// TIA Portal project "DistributionMPS" (V16)

(* hardware
DEVICE "S7-1200 station_1"  S7-1200 Station
   slot 0: "Rack_0"  S7-1200 Rack  Rack  V1.0
   slot 1: "PLC_1"  CPU 1214C AC/DC/Rly  6ES7 214-1BG31-0XB0  V3.0
DEVICE "HMI_1"  KTP600 Basic color PN
   slot 0: "HMI_1"  KTP600 Basic color PN  6AV6 647-0AD11-3AX0  12.0.0.0
   slot 1: "HMI_RT_1"  KTP600 Basic color PN  6AV6 647-0AD11-3AX0  12.0.0.0
   slot 5: "HMI_1.IE_CP_1"  PROFINET Interface  12.0.0.0
      slot 1: "Interfaz PROFINET_1"  PROFINET Interface
         slot 1: "Port_1"  Port
*)

// ===== PLC "PLC_1"  CPU 1214C AC/DC/Rly =====

VAR_GLOBAL   // PLC tag table "Tabla de variables estándar"
   "Conveyor_Forward" AT %Q0.0 : Bool;
   "Conveyor_Reverse" AT %Q0.1 : Bool;
   "Splitter" AT %Q0.2 : Bool;
   "Slider" AT %Q0.4 : Bool;
   "WP_Beg" AT %I0.0 : Bool;
   "WP_Mid" AT %I0.1 : Bool;
   "No_WP_End" AT %I0.2 : Bool;
   "Slider_Init" AT %I0.4 : Bool;
   "Slider_End" AT %I0.5 : Bool;
   "Mag_Empty" AT %I0.6 : Bool;
   "System_Ready" AT %M0.0 : Bool;
   "WP_In" AT %M0.1 : Bool;
   "WP_Eject" AT %M0.2 : Bool;
   "WP_In_Conveyor" AT %M0.3 : Bool;
   "No_WP_In_Mag" AT %M0.4 : Bool;
   "WP_Ej_Conveyor" AT %M0.5 : Bool;
END_VAR

// folder: System blocks/Program resources

DATA_BLOCK "IEC_Timer_0_DB"   // DB1
{ S7_Optimized_Access := 'TRUE' }
AUTHOR : Simatic
FAMILY : IEC
NAME : IEC_TMR
VERSION : 1.0
// stored: InstanceOfName IEC_TIMER
"IEC_TIMER"
BEGIN
END_DATA_BLOCK

DATA_BLOCK "IEC_Timer_0_DB_1"   // DB2
{ S7_Optimized_Access := 'TRUE' }
AUTHOR : Simatic
FAMILY : IEC
NAME : IEC_TMR
VERSION : 1.0
// stored: InstanceOfName IEC_TIMER
"IEC_TIMER"
BEGIN
END_DATA_BLOCK

// folder: (top level)

ORGANIZATION_BLOCK "Main"   // OB1, LAD, ProgramCycle
TITLE = "Main Program Sweep (Cycle)"
{ S7_Optimized_Access := 'TRUE' }
VERSION : 0.1
   VAR_TEMP   // added for the SCL form of the ladder/FBD networks
      _w1 : Bool;
   END_VAR
BEGIN

REGION Network 1: Identificar Pieza
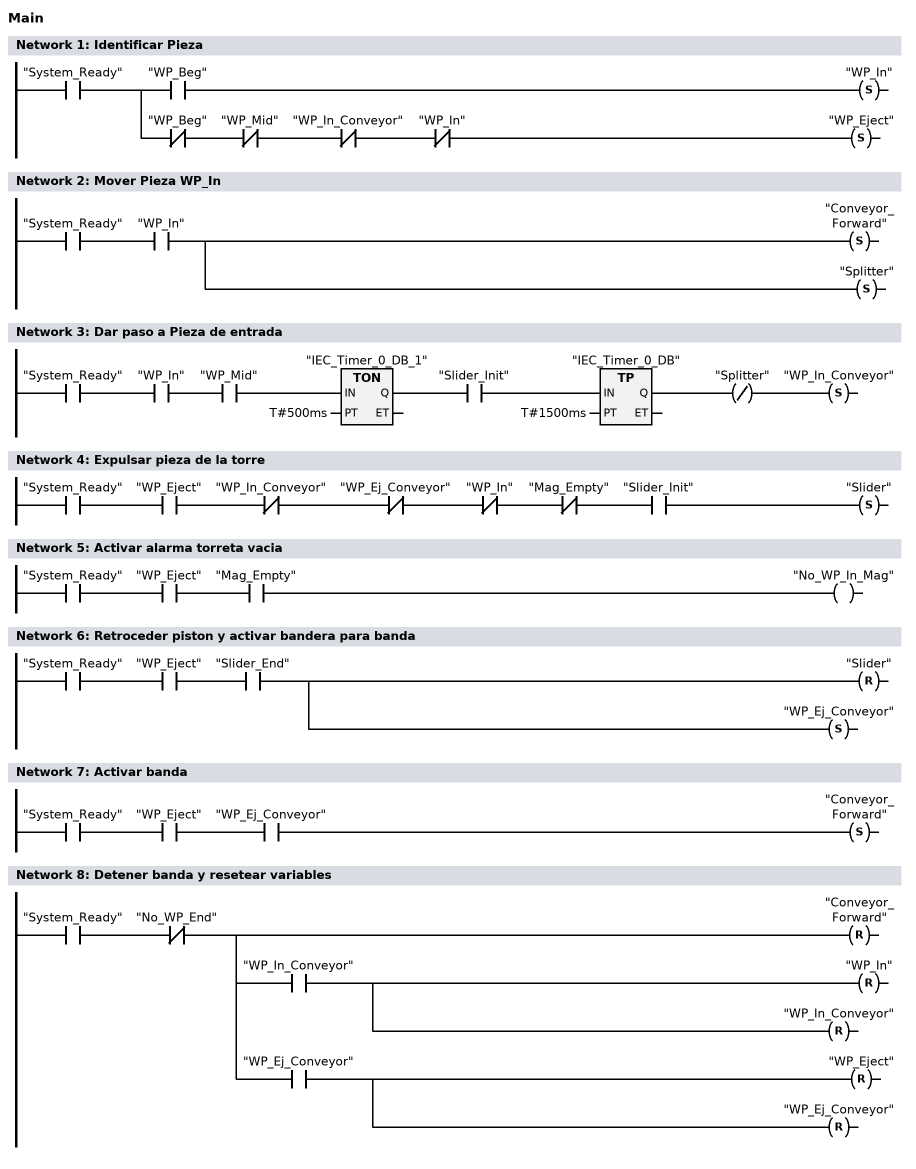
   RUNG wire#powerrail
      Contact( "System_Ready" )
      wire#w1
      Contact( "WP_Beg" )
      S_Coil( "WP_In" )
   END_RUNG
   RUNG wire#w1
      I_Contact( "WP_Beg" )
      I_Contact( "WP_Mid" )
      I_Contact( "WP_In_Conveyor" )
      I_Contact( "WP_In" )
      S_Coil( "WP_Eject" )
   END_RUNG
   // the same network as SCL:
   IF "System_Ready" AND "WP_Beg" THEN "WP_In" := TRUE; END_IF;
   IF "System_Ready" AND NOT "WP_Beg" AND NOT "WP_Mid" AND NOT "WP_In_Conveyor" AND NOT "WP_In" THEN
       "WP_Eject" := TRUE;
   END_IF;
END_REGION

REGION Network 2: Mover Pieza WP_In
   RUNG wire#powerrail
      Contact( "System_Ready" )
      Contact( "WP_In" )
      wire#w1
      S_Coil( "Conveyor_Forward" )
   END_RUNG
   RUNG wire#w1
      S_Coil( "Splitter" )
   END_RUNG
   // the same network as SCL:
   IF "System_Ready" AND "WP_In" THEN
       "Conveyor_Forward" := TRUE;
       "Splitter" := TRUE;
   END_IF;
END_REGION

REGION Network 3: Dar paso a Pieza de entrada
   "IEC_Timer_0_DB_1".TON(IN := "System_Ready" AND "WP_In" AND "WP_Mid", PT := T#500ms);
   "IEC_Timer_0_DB".TP(IN := "IEC_Timer_0_DB_1".Q AND "Slider_Init", PT := T#1500ms);
   "Splitter" := NOT "IEC_Timer_0_DB".Q;
   IF "IEC_Timer_0_DB".Q THEN "WP_In_Conveyor" := TRUE; END_IF;
END_REGION

REGION Network 4: Expulsar pieza de la torre
   RUNG wire#powerrail
      Contact( "System_Ready" )
      Contact( "WP_Eject" )
      I_Contact( "WP_In_Conveyor" )
      I_Contact( "WP_Ej_Conveyor" )
      I_Contact( "WP_In" )
      I_Contact( "Mag_Empty" )
      Contact( "Slider_Init" )
      S_Coil( "Slider" )
   END_RUNG
   // the same network as SCL:
   IF "System_Ready" AND "WP_Eject" AND NOT "WP_In_Conveyor" AND NOT "WP_Ej_Conveyor" AND NOT "WP_In" AND NOT "Mag_Empty" AND "Slider_Init" THEN
       "Slider" := TRUE;
   END_IF;
END_REGION

REGION Network 5: Activar alarma torreta vacia
   RUNG wire#powerrail
      Contact( "System_Ready" )
      Contact( "WP_Eject" )
      Contact( "Mag_Empty" )
      Coil( "No_WP_In_Mag" )
   END_RUNG
   // the same network as SCL:
   "No_WP_In_Mag" := "System_Ready" AND "WP_Eject" AND "Mag_Empty";
END_REGION

REGION Network 6: Retroceder piston y activar bandera para banda
   RUNG wire#powerrail
      Contact( "System_Ready" )
      Contact( "WP_Eject" )
      Contact( "Slider_End" )
      wire#w1
      R_Coil( "Slider" )
   END_RUNG
   RUNG wire#w1
      S_Coil( "WP_Ej_Conveyor" )
   END_RUNG
   // the same network as SCL:
   IF "System_Ready" AND "WP_Eject" AND "Slider_End" THEN
       "Slider" := FALSE;
       "WP_Ej_Conveyor" := TRUE;
   END_IF;
END_REGION

REGION Network 7: Activar banda
   RUNG wire#powerrail
      Contact( "System_Ready" )
      Contact( "WP_Eject" )
      Contact( "WP_Ej_Conveyor" )
      S_Coil( "Conveyor_Forward" )
   END_RUNG
   // the same network as SCL:
   IF "System_Ready" AND "WP_Eject" AND "WP_Ej_Conveyor" THEN "Conveyor_Forward" := TRUE; END_IF;
END_REGION

REGION Network 8: Detener banda y resetear variables
   RUNG wire#powerrail
      Contact( "System_Ready" )
      I_Contact( "No_WP_End" )
      wire#w1
      R_Coil( "Conveyor_Forward" )
   END_RUNG
   RUNG wire#w1
      Contact( "WP_In_Conveyor" )
      wire#w2
      R_Coil( "WP_In" )
   END_RUNG
   RUNG wire#w2
      R_Coil( "WP_In_Conveyor" )
   END_RUNG
   RUNG wire#w1
      Contact( "WP_Ej_Conveyor" )
      wire#w3
      R_Coil( "WP_Eject" )
   END_RUNG
   RUNG wire#w3
      R_Coil( "WP_Ej_Conveyor" )
   END_RUNG
   // the same network as SCL:
   #_w1 := "System_Ready" AND NOT "No_WP_End";
   IF #_w1 THEN "Conveyor_Forward" := FALSE; END_IF;
   IF #_w1 AND "WP_In_Conveyor" THEN
       "WP_In" := FALSE;
       "WP_In_Conveyor" := FALSE;
   END_IF;
   IF #_w1 AND "WP_Ej_Conveyor" THEN
       "WP_Eject" := FALSE;
       "WP_Ej_Conveyor" := FALSE;
   END_IF;
END_REGION
END_ORGANIZATION_BLOCK

ORGANIZATION_BLOCK "Startup"   // OB100, LAD, Startup
TITLE = "Complete Restart"
{ S7_Optimized_Access := 'TRUE' }
VERSION : 0.1
   VAR_INPUT
      LostRetentive : Bool;   // True if retentive data are lost
      LostRTC : Bool;   // True if date and time are lost
   END_VAR
BEGIN

REGION Network 1
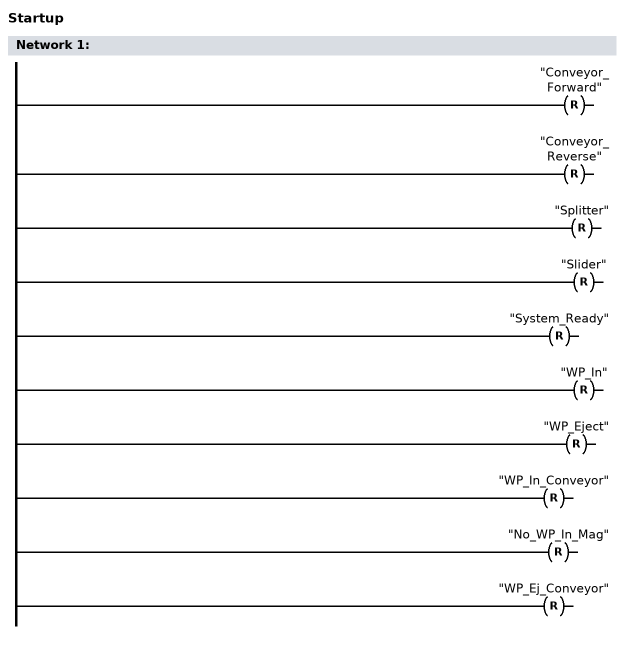
   RUNG wire#powerrail
      R_Coil( "Conveyor_Forward" )
   END_RUNG
   RUNG wire#powerrail
      R_Coil( "Conveyor_Reverse" )
   END_RUNG
   RUNG wire#powerrail
      R_Coil( "Splitter" )
   END_RUNG
   RUNG wire#powerrail
      R_Coil( "Slider" )
   END_RUNG
   RUNG wire#powerrail
      R_Coil( "System_Ready" )
   END_RUNG
   RUNG wire#powerrail
      R_Coil( "WP_In" )
   END_RUNG
   RUNG wire#powerrail
      R_Coil( "WP_Eject" )
   END_RUNG
   RUNG wire#powerrail
      R_Coil( "WP_In_Conveyor" )
   END_RUNG
   RUNG wire#powerrail
      R_Coil( "No_WP_In_Mag" )
   END_RUNG
   RUNG wire#powerrail
      R_Coil( "WP_Ej_Conveyor" )
   END_RUNG
   // the same network as SCL:
   "Conveyor_Forward" := FALSE;
   "Conveyor_Reverse" := FALSE;
   "Splitter" := FALSE;
   "Slider" := FALSE;
   "System_Ready" := FALSE;
   "WP_In" := FALSE;
   "WP_Eject" := FALSE;
   "WP_In_Conveyor" := FALSE;
   "No_WP_In_Mag" := FALSE;
   "WP_Ej_Conveyor" := FALSE;
END_REGION
END_ORGANIZATION_BLOCK

(* ===== HMI "HMI_RT_1" =====
system functions are stored by id; their names below are inferred from use
connection "HMI_Conexión_1": ETHERNET, SMART_S7_1200_OMS

HMI tags "Tabla de variables estándar"
   "Número_imagen_variable" : UInt, internal
   "System_Ready" : Bool = PLC System_Ready AT %M0.0, 1 s

text list "Nombre_imagen_lista_texto": 1 'Imagen raíz'; 2 'Imagen0'; 3 'Imagen1'; 4 'Imágenes de sistema'; 5 'Diagnóstico de sistema SIMATIC PLC'; 6 'Información del proyecto'

screen "Información del proyecto" 320x240, template "Plantilla_1"
   on GenerateScreen: SetTag("Número_imagen_variable", 6)
   TextField "HmiScreenItemData" at 4,71 size 120x20; Text 'Nombre del proyecto:'
   TextField "HmiScreenItemData_1" at 128,71 size 188x20; Text 'DistributionMPS'
   TextField "HmiScreenItemData_2" at 4,92 size 120x20; Text 'Creado:'
   TextField "HmiScreenItemData_3" at 128,92 size 188x20; Text '14/02/2022 11:56:09'
   TextField "HmiScreenItemData_4" at 4,113 size 120x20; Text 'Autor:'
   TextField "HmiScreenItemData_5" at 128,113 size 188x20; Text 'Robotrifasicos'
   TextField "HmiScreenItemData_6" at 4,134 size 120x20; Text 'Descripción:'
   TextField "HmiScreenItemData_7" at 128,134 size 188x20; Text '(no configurado)'
   Button "Atrás" at 1,39 size 104x30; TextOff 'Atrás'
      on Release: ActivateScreen("Imágenes de sistema", 0)

Template "Plantilla_1" 320x240
   Button "Salir" at 266,202 size 52x37; TextOff 'Salir'; PictureOff "ExitRuntime_KTP600_Basic_color_PN"; PictureOn "ExitRuntime_KTP600_Basic_color_PN"
      on Release: StopRuntime(0)
   Button "Template_Button" at 213,202 size 52x37; TextOff 'Text'
   Button "Template_Button_1" at 160,202 size 52x37; TextOff 'Text'
   Button "Template_Button_2" at 107,202 size 52x37; TextOff 'Text'
   Button "Avisos" at 54,202 size 52x37; TextOff 'Avisos'; PictureOff "AlarmDisplay_KTP600_Basic_color_PN"; PictureOn "AlarmDisplay_KTP600_Basic_color_PN"
      on Release: function_ef3f5d25("Ventana de avisos_no_acusado", -1)
   Button "Imagen inicial" at 1,202 size 52x37; TextOff 'Imagen inicial'; PictureOff "NavigateHome_KTP600_Basic_color_PN"; PictureOn "NavigateHome_KTP600_Basic_color_PN"
      on Release: ActivateScreen("Imagen raíz", 0)
   SymbolicIOField "Imagen_campo_ES_simbólico" at 69,7 size 164x24; TextOff '0'; TextOn '1'; TextList "Nombre_imagen_lista_texto"
      ProcessValue <- "Número_imagen_variable"
      on Change: ActivateScreenByNumber("Número_imagen_variable", 0)
   DateTimeField "HmiScreenItemData" at 235,19 size 85x19
   DateTimeField "HmiScreenItemData_1" at 235,0 size 85x19
   GraphicView "Logotipo" at 0,0 size 67x38; Picture "Logotipo de HMI_1"

screen "Imagen raíz" 320x240, template "Plantilla_1"
   on GenerateScreen: SetTag("Número_imagen_variable", 1)
   Button "Imágenes de sistema" at 211,39 size 104x30; TextOff 'Imágenes de sis...'
      on Release: ActivateScreen("Imágenes de sistema", 0)
   Button "Botón_1" at 15,88 size 96x32; TextOff 'Start'
      on Press: SetBit("System_Ready")
   Button "Botón_2" at 204,88 size 96x32; TextOff 'Stop'
      on Press: ResetBit("System_Ready")
   TextField "Text field_1" at 16,157 size 111x35; Text 'Por: Felipe Arenas Uribe Diego Lopez Guerrero'

screen "Imágenes de sistema" 320x240, template "Plantilla_1"
   on GenerateScreen: SetTag("Número_imagen_variable", 4)
   TextField "HmiScreenItemData" at 32,109 size 256x17; Text 'Imágenes de sistema'
   Button "Atrás" at 1,39 size 104x30; TextOff 'Atrás'
      on Release: ActivateScreen("Imagen raíz", 0)
   Button "Diagnóstico de sistema SIMATIC PLC" at 106,39 size 104x30; TextOff 'Diagnóstico de ...'
      on Release: ActivateScreen("Diagnóstico de sistema SIMATIC PLC", 0)
   Button "Información del proyecto" at 211,39 size 104x30; TextOff 'Información del ...'
      on Release: ActivateScreen("Información del proyecto", 0)

screen "Diagnóstico de sistema SIMATIC PLC" 320x240, template "Plantilla_1"
   on GenerateScreen: SetTag("Número_imagen_variable", 5)
   SysDiagControl "HmiScreenItemData" at 1,70 size 316x125
   Button "Atrás" at 1,39 size 104x30; TextOff 'Atrás'
      on Release: ActivateScreen("Imágenes de sistema", 0)
*)